PROGRAM PRG_PMPS
VAR
 fbArbiterIO : FB_SubSysToArbiter_IO;
 test : bool;
END_VAR

(*Fast Fault instantiation*)
g_FastFaultOutput1.bAutoReset :=TRUE;
g_FastFaultOutput2.bAutoReset :=TRUE;
g_FastFaultOutput1.Execute();
g_FastFaultOutput2.Execute();


(* Arbiter Instantiation*)
(*Arbiter one responsible for the aperture valves*)
fbArbiterIO(Arbiter := GVL_ILK.g_fbArbiter, fbFFHWO := GVL_ILK.g_FastFaultOutput1);

//test := GVL_ILK.g_fbArbiter.CheckRequest(1001);


test := GVL_ILK.g_fbArbiter.CheckRequestInPool(1001);

END_PROGRAM

(* stored: Version 1.1.0.1, ProductVersion 3.1.4022.18
   POU PRG_PMPS: Id {3bbd9cd5-72c9-4b35-aa2f-63d3e3610a6e}, SpecialFunc None *)
